// Block: TEST_Production

DATA_BLOCK TEST_Production
VERSION : 0.1
   NON_RETAIN
   VAR
      O_ACT : Struct
         ABILITA_FC : Bool;
         RETVAL : DInt;
         Push : Bool;
         Pop : Bool;
         Pop_To_TODO : Bool;
         Pop_To_ENDING : Bool;
         Ordine : Prod_Item;
      END_STRUCT;
      O_TODO : Struct
         ABILITA_FC : Bool;
         RETVAL : DInt;
         Clear_Gap : Bool;
         Push_Top : Bool;
         Push_Bottom : Bool;
         Pop : Bool;
         Pop_Index : Int;
         "Pop_&_Push_ACT" : Bool;
         "Pop_&_Push_ENDING" : Bool;
         Evaluate_FULL : Bool;
         Ordine : Prod_Item;
      END_STRUCT;
      O_ENDING : Struct
         ABILITA_FC : Bool;
         RETVAL : DInt;
         Index : Int;
         Clear_Gap : Bool;
         Push_Top : Bool;
         Pop : Bool;
         "Pop_&_O_OUT_Push" : Bool;
         "Pop_&_O_TODO_Push" : Bool;
         Ordine : Prod_Item;
      END_STRUCT;
      O_OUT : Struct
         ABILITA_FC : Bool;
         RETVAL : DInt;
         Index : Int;
         Clear_Gap : Bool;
         Push_Top : Bool;
         Pop : Bool;
         Ordine : Prod_Item;
      END_STRUCT;
      O_ENDING_Cleaning : Struct
         Enable : Bool;
         AckChangeStep : Bool;
         ActualStep : Int;
      END_STRUCT;
   END_VAR

BEGIN
   // No initialization required
END_DATA_BLOCK
